// TIA Portal V21 export
VAR_GLOBAL   // PLC tag table "Default tag table"
END_VAR
